(* PLC project EXAMPLE_MOD, Beckhoff Automation GmbH TwinCAT PLC Control 3.5.13.20 *)
(* stored: creationDateTime 2020-06-22T11:49:20.3012497, modificationDateTime 2020-06-22T11:49:20.3012497 *)

PROGRAM POU
VAR
	A: BOOL;
	B: BOOL;
	C: BOOL;
END_VAR

            
IF (A) THEN 
	B := FALSE;
	C := TRUE;
END_IF
          
END_PROGRAM
